{attribute 'qualified_only'}
VAR_GLOBAL CONSTANT
	FalseValue : FalseBoolValue := ();
	TrueValue : TrueBoolValue := ();
END_VAR

(* stored: Version 1.1.0.1
   GVL BoolValues: Id {fbfbab9c-b9e2-45c2-963b-b3aa3b72aad8} *)
